FUNCTION_BLOCK FB_Toggle2Tap
///////////
// FB to change a toggle into a tap with constant duration//
///////////

VAR_INPUT
	TapDuration		: TIME; 	// (s) Tap duration
	
	ToggleVar 		: BOOL;		// Toggled input variable 

	
END_VAR

VAR_OUTPUT
	TapVar			: BOOL ; 	// Tapped output variable
	
END_VAR

VAR				
	R_TRIG			: R_TRIG ;				// Create a square at Rising Edge Detection
	F_TRIG			: F_TRIG ;				// Create a square at falling Edge Detection 
	TP				: TP ; 					// Square Signal 

END_VAR

R_TRIG(CLK := ToggleVar) ;  							// Rising Edge Detection
F_TRIG(CLK := ToggleVar) ; 								// Falling Edge Detection

TP(IN := R_TRIG.Q OR F_TRIG.Q , PT := TapDuration) ;  	// Square signal 

TapVar		:= TP.Q ; 									// OUtput variable

END_FUNCTION_BLOCK

(* stored: Version 1.1.0.1, ProductVersion 3.1.4024.6
   POU FB_Toggle2Tap: Id {5816cccc-b91f-421a-9ef2-a8a78c3771e3}, SpecialFunc None *)
